// TIA Portal V18 export
// export: Created 2026-06-07T17:38:18.1714676Z, ExportSetting WithDefaults, DisplayName Totally Integrated Automation Portal, DisplayVersion V18, DisplayName TIA Portal Openness, DisplayVersion V18, DisplayName TIA Portal Version Control Interface, DisplayVersion V18, DisplayName STEP 7 Professional, DisplayVersion V18, DisplayName STEP 7 Safety, DisplayVersion V18, DisplayName WinCC Professional, DisplayVersion V18
FUNCTION "FC_HMI_Mirror_PLC1" : Void   // FC41, LAD
{ S7_Optimized_Access := 'TRUE' }
VERSION : 0.1
// stored: AutoNumber true, IsIECCheckEnabled false, SetENOAutomatically false, UDAEnableTagReadback false
BEGIN

REGION Network 1: Mirror AI_V3230_Nuoc_Bon1
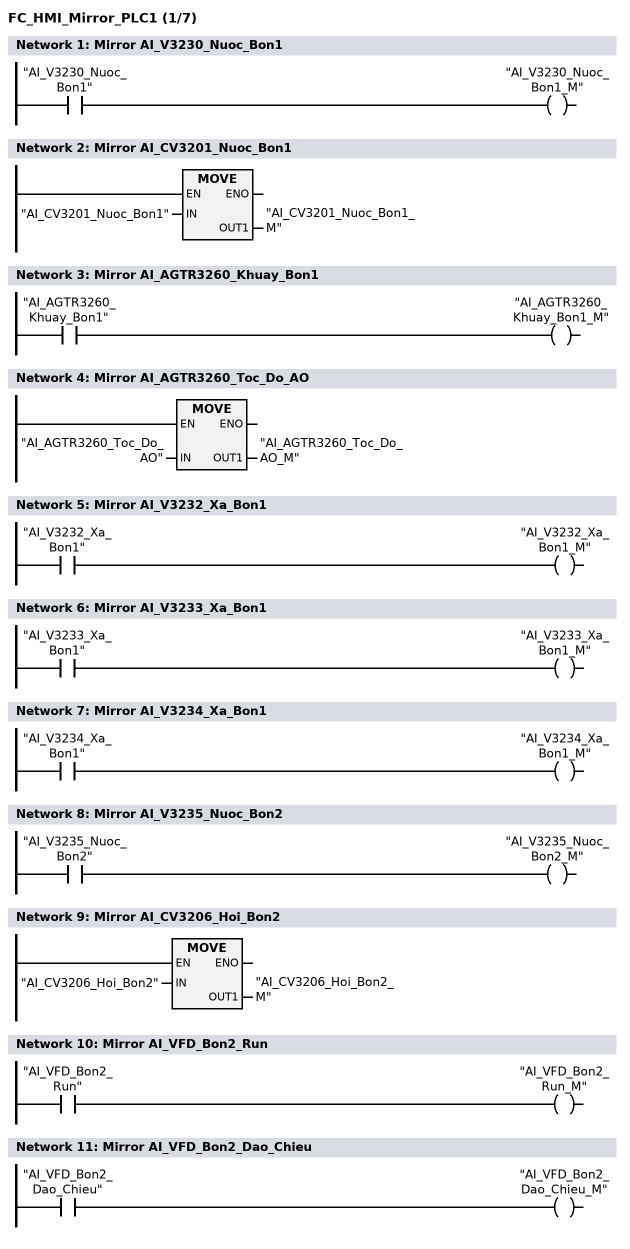
   RUNG wire#powerrail
      Contact( "AI_V3230_Nuoc_Bon1" )
      Coil( "AI_V3230_Nuoc_Bon1_M" )
   END_RUNG
   // the same network as SCL:
   "AI_V3230_Nuoc_Bon1_M" := "AI_V3230_Nuoc_Bon1";
END_REGION

REGION Network 2: Mirror AI_CV3201_Nuoc_Bon1
   RUNG wire#powerrail
      { S7_GenerateENO := "TRUE" } Move(in := "AI_CV3201_Nuoc_Bon1", out1 => "AI_CV3201_Nuoc_Bon1_M")
   END_RUNG
   // the same network as SCL:
   "AI_CV3201_Nuoc_Bon1_M" := "AI_CV3201_Nuoc_Bon1";
END_REGION

REGION Network 3: Mirror AI_AGTR3260_Khuay_Bon1
   RUNG wire#powerrail
      Contact( "AI_AGTR3260_Khuay_Bon1" )
      Coil( "AI_AGTR3260_Khuay_Bon1_M" )
   END_RUNG
   // the same network as SCL:
   "AI_AGTR3260_Khuay_Bon1_M" := "AI_AGTR3260_Khuay_Bon1";
END_REGION

REGION Network 4: Mirror AI_AGTR3260_Toc_Do_AO
   RUNG wire#powerrail
      { S7_GenerateENO := "TRUE" } Move(in := "AI_AGTR3260_Toc_Do_AO", out1 => "AI_AGTR3260_Toc_Do_AO_M")
   END_RUNG
   // the same network as SCL:
   "AI_AGTR3260_Toc_Do_AO_M" := "AI_AGTR3260_Toc_Do_AO";
END_REGION

REGION Network 5: Mirror AI_V3232_Xa_Bon1
   RUNG wire#powerrail
      Contact( "AI_V3232_Xa_Bon1" )
      Coil( "AI_V3232_Xa_Bon1_M" )
   END_RUNG
   // the same network as SCL:
   "AI_V3232_Xa_Bon1_M" := "AI_V3232_Xa_Bon1";
END_REGION

REGION Network 6: Mirror AI_V3233_Xa_Bon1
   RUNG wire#powerrail
      Contact( "AI_V3233_Xa_Bon1" )
      Coil( "AI_V3233_Xa_Bon1_M" )
   END_RUNG
   // the same network as SCL:
   "AI_V3233_Xa_Bon1_M" := "AI_V3233_Xa_Bon1";
END_REGION

REGION Network 7: Mirror AI_V3234_Xa_Bon1
   RUNG wire#powerrail
      Contact( "AI_V3234_Xa_Bon1" )
      Coil( "AI_V3234_Xa_Bon1_M" )
   END_RUNG
   // the same network as SCL:
   "AI_V3234_Xa_Bon1_M" := "AI_V3234_Xa_Bon1";
END_REGION

REGION Network 8: Mirror AI_V3235_Nuoc_Bon2
   RUNG wire#powerrail
      Contact( "AI_V3235_Nuoc_Bon2" )
      Coil( "AI_V3235_Nuoc_Bon2_M" )
   END_RUNG
   // the same network as SCL:
   "AI_V3235_Nuoc_Bon2_M" := "AI_V3235_Nuoc_Bon2";
END_REGION

REGION Network 9: Mirror AI_CV3206_Hoi_Bon2
   RUNG wire#powerrail
      { S7_GenerateENO := "TRUE" } Move(in := "AI_CV3206_Hoi_Bon2", out1 => "AI_CV3206_Hoi_Bon2_M")
   END_RUNG
   // the same network as SCL:
   "AI_CV3206_Hoi_Bon2_M" := "AI_CV3206_Hoi_Bon2";
END_REGION

REGION Network 10: Mirror AI_VFD_Bon2_Run
   RUNG wire#powerrail
      Contact( "AI_VFD_Bon2_Run" )
      Coil( "AI_VFD_Bon2_Run_M" )
   END_RUNG
   // the same network as SCL:
   "AI_VFD_Bon2_Run_M" := "AI_VFD_Bon2_Run";
END_REGION

REGION Network 11: Mirror AI_VFD_Bon2_Dao_Chieu
   RUNG wire#powerrail
      Contact( "AI_VFD_Bon2_Dao_Chieu" )
      Coil( "AI_VFD_Bon2_Dao_Chieu_M" )
   END_RUNG
   // the same network as SCL:
   "AI_VFD_Bon2_Dao_Chieu_M" := "AI_VFD_Bon2_Dao_Chieu";
END_REGION

REGION Network 12: Mirror AI_VFD_Bon2_Toc_Do_AO
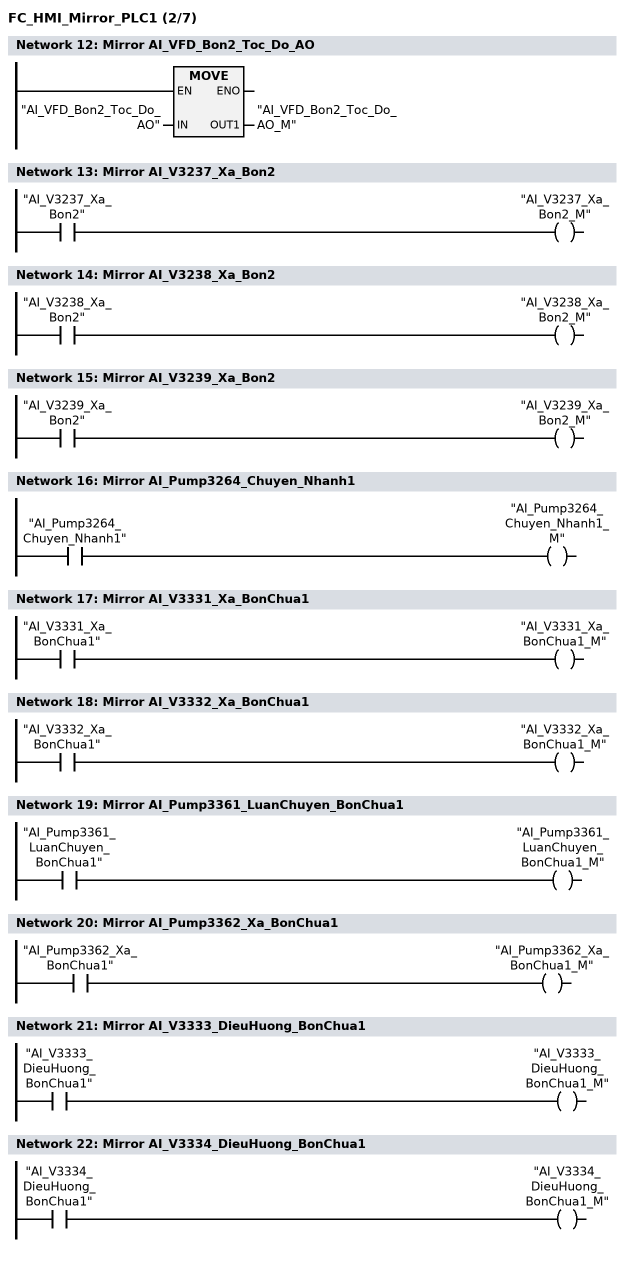
   RUNG wire#powerrail
      { S7_GenerateENO := "TRUE" } Move(in := "AI_VFD_Bon2_Toc_Do_AO", out1 => "AI_VFD_Bon2_Toc_Do_AO_M")
   END_RUNG
   // the same network as SCL:
   "AI_VFD_Bon2_Toc_Do_AO_M" := "AI_VFD_Bon2_Toc_Do_AO";
END_REGION

REGION Network 13: Mirror AI_V3237_Xa_Bon2
   RUNG wire#powerrail
      Contact( "AI_V3237_Xa_Bon2" )
      Coil( "AI_V3237_Xa_Bon2_M" )
   END_RUNG
   // the same network as SCL:
   "AI_V3237_Xa_Bon2_M" := "AI_V3237_Xa_Bon2";
END_REGION

REGION Network 14: Mirror AI_V3238_Xa_Bon2
   RUNG wire#powerrail
      Contact( "AI_V3238_Xa_Bon2" )
      Coil( "AI_V3238_Xa_Bon2_M" )
   END_RUNG
   // the same network as SCL:
   "AI_V3238_Xa_Bon2_M" := "AI_V3238_Xa_Bon2";
END_REGION

REGION Network 15: Mirror AI_V3239_Xa_Bon2
   RUNG wire#powerrail
      Contact( "AI_V3239_Xa_Bon2" )
      Coil( "AI_V3239_Xa_Bon2_M" )
   END_RUNG
   // the same network as SCL:
   "AI_V3239_Xa_Bon2_M" := "AI_V3239_Xa_Bon2";
END_REGION

REGION Network 16: Mirror AI_Pump3264_Chuyen_Nhanh1
   RUNG wire#powerrail
      Contact( "AI_Pump3264_Chuyen_Nhanh1" )
      Coil( "AI_Pump3264_Chuyen_Nhanh1_M" )
   END_RUNG
   // the same network as SCL:
   "AI_Pump3264_Chuyen_Nhanh1_M" := "AI_Pump3264_Chuyen_Nhanh1";
END_REGION

REGION Network 17: Mirror AI_V3331_Xa_BonChua1
   RUNG wire#powerrail
      Contact( "AI_V3331_Xa_BonChua1" )
      Coil( "AI_V3331_Xa_BonChua1_M" )
   END_RUNG
   // the same network as SCL:
   "AI_V3331_Xa_BonChua1_M" := "AI_V3331_Xa_BonChua1";
END_REGION

REGION Network 18: Mirror AI_V3332_Xa_BonChua1
   RUNG wire#powerrail
      Contact( "AI_V3332_Xa_BonChua1" )
      Coil( "AI_V3332_Xa_BonChua1_M" )
   END_RUNG
   // the same network as SCL:
   "AI_V3332_Xa_BonChua1_M" := "AI_V3332_Xa_BonChua1";
END_REGION

REGION Network 19: Mirror AI_Pump3361_LuanChuyen_BonChua1
   RUNG wire#powerrail
      Contact( "AI_Pump3361_LuanChuyen_BonChua1" )
      Coil( "AI_Pump3361_LuanChuyen_BonChua1_M" )
   END_RUNG
   // the same network as SCL:
   "AI_Pump3361_LuanChuyen_BonChua1_M" := "AI_Pump3361_LuanChuyen_BonChua1";
END_REGION

REGION Network 20: Mirror AI_Pump3362_Xa_BonChua1
   RUNG wire#powerrail
      Contact( "AI_Pump3362_Xa_BonChua1" )
      Coil( "AI_Pump3362_Xa_BonChua1_M" )
   END_RUNG
   // the same network as SCL:
   "AI_Pump3362_Xa_BonChua1_M" := "AI_Pump3362_Xa_BonChua1";
END_REGION

REGION Network 21: Mirror AI_V3333_DieuHuong_BonChua1
   RUNG wire#powerrail
      Contact( "AI_V3333_DieuHuong_BonChua1" )
      Coil( "AI_V3333_DieuHuong_BonChua1_M" )
   END_RUNG
   // the same network as SCL:
   "AI_V3333_DieuHuong_BonChua1_M" := "AI_V3333_DieuHuong_BonChua1";
END_REGION

REGION Network 22: Mirror AI_V3334_DieuHuong_BonChua1
   RUNG wire#powerrail
      Contact( "AI_V3334_DieuHuong_BonChua1" )
      Coil( "AI_V3334_DieuHuong_BonChua1_M" )
   END_RUNG
   // the same network as SCL:
   "AI_V3334_DieuHuong_BonChua1_M" := "AI_V3334_DieuHuong_BonChua1";
END_REGION

REGION Network 23: Mirror AI_V3335_DieuHuong_BonChua1
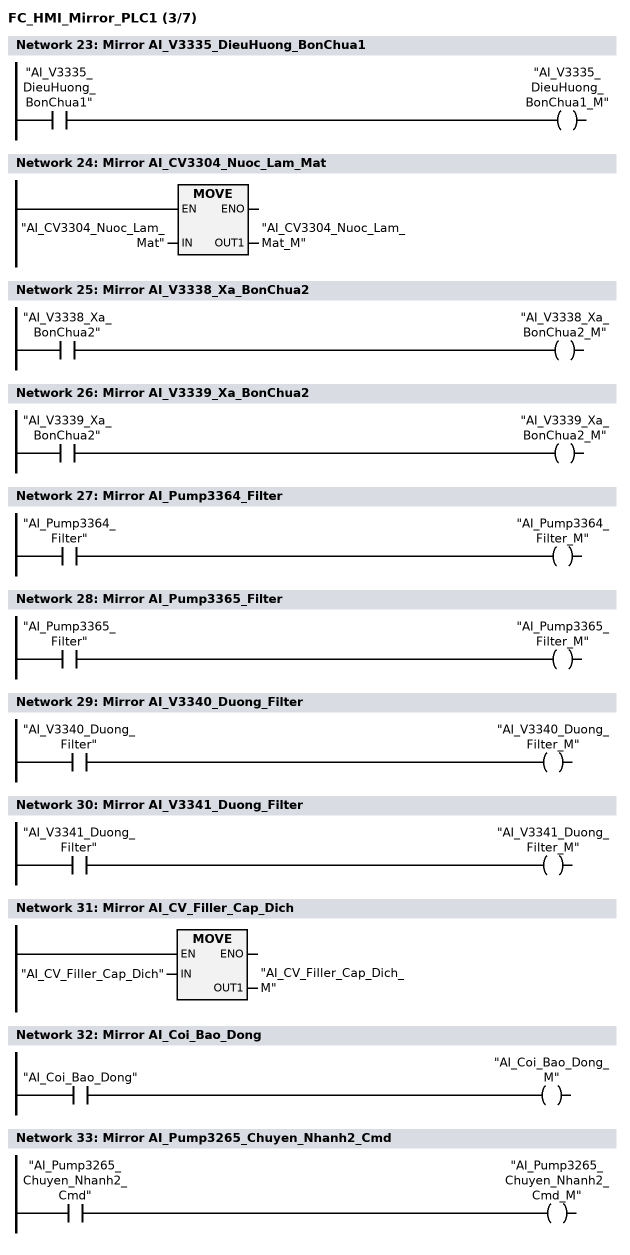
   RUNG wire#powerrail
      Contact( "AI_V3335_DieuHuong_BonChua1" )
      Coil( "AI_V3335_DieuHuong_BonChua1_M" )
   END_RUNG
   // the same network as SCL:
   "AI_V3335_DieuHuong_BonChua1_M" := "AI_V3335_DieuHuong_BonChua1";
END_REGION

REGION Network 24: Mirror AI_CV3304_Nuoc_Lam_Mat
   RUNG wire#powerrail
      { S7_GenerateENO := "TRUE" } Move(in := "AI_CV3304_Nuoc_Lam_Mat", out1 => "AI_CV3304_Nuoc_Lam_Mat_M")
   END_RUNG
   // the same network as SCL:
   "AI_CV3304_Nuoc_Lam_Mat_M" := "AI_CV3304_Nuoc_Lam_Mat";
END_REGION

REGION Network 25: Mirror AI_V3338_Xa_BonChua2
   RUNG wire#powerrail
      Contact( "AI_V3338_Xa_BonChua2" )
      Coil( "AI_V3338_Xa_BonChua2_M" )
   END_RUNG
   // the same network as SCL:
   "AI_V3338_Xa_BonChua2_M" := "AI_V3338_Xa_BonChua2";
END_REGION

REGION Network 26: Mirror AI_V3339_Xa_BonChua2
   RUNG wire#powerrail
      Contact( "AI_V3339_Xa_BonChua2" )
      Coil( "AI_V3339_Xa_BonChua2_M" )
   END_RUNG
   // the same network as SCL:
   "AI_V3339_Xa_BonChua2_M" := "AI_V3339_Xa_BonChua2";
END_REGION

REGION Network 27: Mirror AI_Pump3364_Filter
   RUNG wire#powerrail
      Contact( "AI_Pump3364_Filter" )
      Coil( "AI_Pump3364_Filter_M" )
   END_RUNG
   // the same network as SCL:
   "AI_Pump3364_Filter_M" := "AI_Pump3364_Filter";
END_REGION

REGION Network 28: Mirror AI_Pump3365_Filter
   RUNG wire#powerrail
      Contact( "AI_Pump3365_Filter" )
      Coil( "AI_Pump3365_Filter_M" )
   END_RUNG
   // the same network as SCL:
   "AI_Pump3365_Filter_M" := "AI_Pump3365_Filter";
END_REGION

REGION Network 29: Mirror AI_V3340_Duong_Filter
   RUNG wire#powerrail
      Contact( "AI_V3340_Duong_Filter" )
      Coil( "AI_V3340_Duong_Filter_M" )
   END_RUNG
   // the same network as SCL:
   "AI_V3340_Duong_Filter_M" := "AI_V3340_Duong_Filter";
END_REGION

REGION Network 30: Mirror AI_V3341_Duong_Filter
   RUNG wire#powerrail
      Contact( "AI_V3341_Duong_Filter" )
      Coil( "AI_V3341_Duong_Filter_M" )
   END_RUNG
   // the same network as SCL:
   "AI_V3341_Duong_Filter_M" := "AI_V3341_Duong_Filter";
END_REGION

REGION Network 31: Mirror AI_CV_Filler_Cap_Dich
   RUNG wire#powerrail
      { S7_GenerateENO := "TRUE" } Move(in := "AI_CV_Filler_Cap_Dich", out1 => "AI_CV_Filler_Cap_Dich_M")
   END_RUNG
   // the same network as SCL:
   "AI_CV_Filler_Cap_Dich_M" := "AI_CV_Filler_Cap_Dich";
END_REGION

REGION Network 32: Mirror AI_Coi_Bao_Dong
   RUNG wire#powerrail
      Contact( "AI_Coi_Bao_Dong" )
      Coil( "AI_Coi_Bao_Dong_M" )
   END_RUNG
   // the same network as SCL:
   "AI_Coi_Bao_Dong_M" := "AI_Coi_Bao_Dong";
END_REGION

REGION Network 33: Mirror AI_Pump3265_Chuyen_Nhanh2_Cmd
   RUNG wire#powerrail
      Contact( "AI_Pump3265_Chuyen_Nhanh2_Cmd" )
      Coil( "AI_Pump3265_Chuyen_Nhanh2_Cmd_M" )
   END_RUNG
   // the same network as SCL:
   "AI_Pump3265_Chuyen_Nhanh2_Cmd_M" := "AI_Pump3265_Chuyen_Nhanh2_Cmd";
END_REGION

REGION Network 34: Mirror AI_VFD_Bon2_Actual_Speed_Feedback
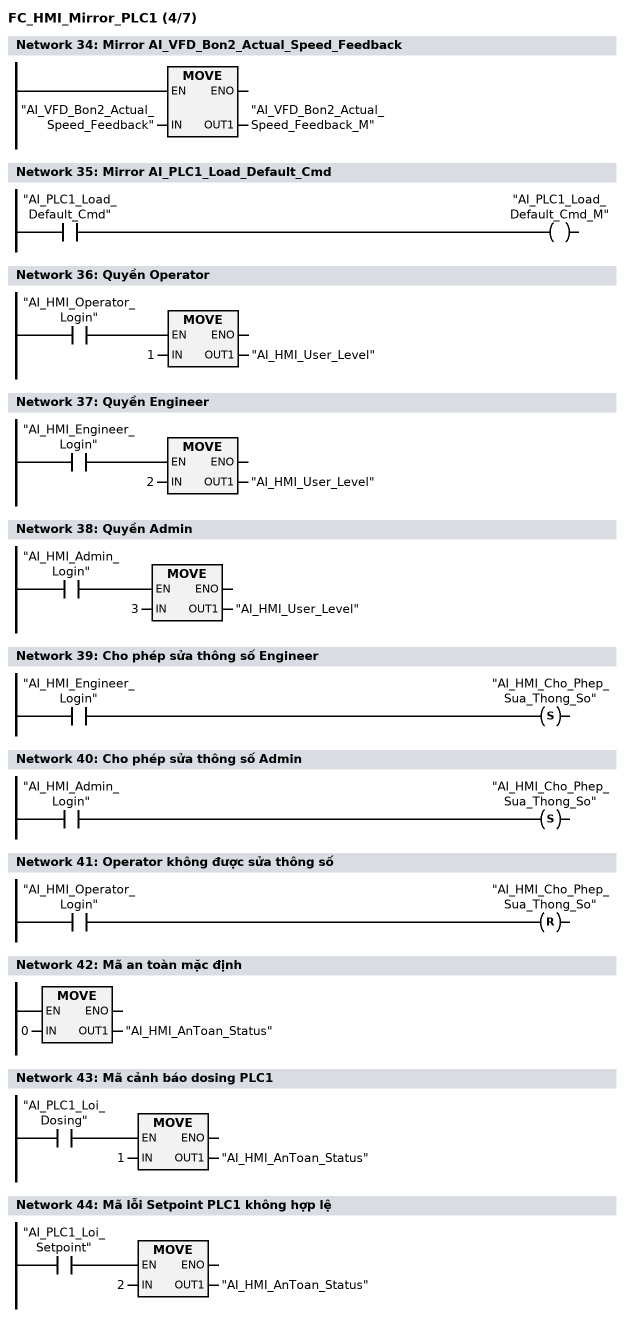
   RUNG wire#powerrail
      { S7_GenerateENO := "TRUE" } Move(in := "AI_VFD_Bon2_Actual_Speed_Feedback", out1 => "AI_VFD_Bon2_Actual_Speed_Feedback_M")
   END_RUNG
   // the same network as SCL:
   "AI_VFD_Bon2_Actual_Speed_Feedback_M" := "AI_VFD_Bon2_Actual_Speed_Feedback";
END_REGION

REGION Network 35: Mirror AI_PLC1_Load_Default_Cmd
   RUNG wire#powerrail
      Contact( "AI_PLC1_Load_Default_Cmd" )
      Coil( "AI_PLC1_Load_Default_Cmd_M" )
   END_RUNG
   // the same network as SCL:
   "AI_PLC1_Load_Default_Cmd_M" := "AI_PLC1_Load_Default_Cmd";
END_REGION

REGION Network 36: Quyền Operator
   RUNG wire#powerrail
      Contact( "AI_HMI_Operator_Login" )
      { S7_GenerateENO := "TRUE" } Move(in := 1, out1 => "AI_HMI_User_Level")
   END_RUNG
   // the same network as SCL:
   IF "AI_HMI_Operator_Login" THEN "AI_HMI_User_Level" := 1; END_IF;
END_REGION

REGION Network 37: Quyền Engineer
   RUNG wire#powerrail
      Contact( "AI_HMI_Engineer_Login" )
      { S7_GenerateENO := "TRUE" } Move(in := 2, out1 => "AI_HMI_User_Level")
   END_RUNG
   // the same network as SCL:
   IF "AI_HMI_Engineer_Login" THEN "AI_HMI_User_Level" := 2; END_IF;
END_REGION

REGION Network 38: Quyền Admin
   RUNG wire#powerrail
      Contact( "AI_HMI_Admin_Login" )
      { S7_GenerateENO := "TRUE" } Move(in := 3, out1 => "AI_HMI_User_Level")
   END_RUNG
   // the same network as SCL:
   IF "AI_HMI_Admin_Login" THEN "AI_HMI_User_Level" := 3; END_IF;
END_REGION

REGION Network 39: Cho phép sửa thông số Engineer
   RUNG wire#powerrail
      Contact( "AI_HMI_Engineer_Login" )
      S_Coil( "AI_HMI_Cho_Phep_Sua_Thong_So" )
   END_RUNG
   // the same network as SCL:
   IF "AI_HMI_Engineer_Login" THEN "AI_HMI_Cho_Phep_Sua_Thong_So" := TRUE; END_IF;
END_REGION

REGION Network 40: Cho phép sửa thông số Admin
   RUNG wire#powerrail
      Contact( "AI_HMI_Admin_Login" )
      S_Coil( "AI_HMI_Cho_Phep_Sua_Thong_So" )
   END_RUNG
   // the same network as SCL:
   IF "AI_HMI_Admin_Login" THEN "AI_HMI_Cho_Phep_Sua_Thong_So" := TRUE; END_IF;
END_REGION

REGION Network 41: Operator không được sửa thông số
   RUNG wire#powerrail
      Contact( "AI_HMI_Operator_Login" )
      R_Coil( "AI_HMI_Cho_Phep_Sua_Thong_So" )
   END_RUNG
   // the same network as SCL:
   IF "AI_HMI_Operator_Login" THEN "AI_HMI_Cho_Phep_Sua_Thong_So" := FALSE; END_IF;
END_REGION

REGION Network 42: Mã an toàn mặc định
   RUNG wire#powerrail
      { S7_GenerateENO := "TRUE" } Move(in := 0, out1 => "AI_HMI_AnToan_Status")
   END_RUNG
   // the same network as SCL:
   "AI_HMI_AnToan_Status" := 0;
END_REGION

REGION Network 43: Mã cảnh báo dosing PLC1
   RUNG wire#powerrail
      Contact( "AI_PLC1_Loi_Dosing" )
      { S7_GenerateENO := "TRUE" } Move(in := 1, out1 => "AI_HMI_AnToan_Status")
   END_RUNG
   // the same network as SCL:
   IF "AI_PLC1_Loi_Dosing" THEN "AI_HMI_AnToan_Status" := 1; END_IF;
END_REGION

REGION Network 44: Mã lỗi Setpoint PLC1 không hợp lệ
   RUNG wire#powerrail
      Contact( "AI_PLC1_Loi_Setpoint" )
      { S7_GenerateENO := "TRUE" } Move(in := 2, out1 => "AI_HMI_AnToan_Status")
   END_RUNG
   // the same network as SCL:
   IF "AI_PLC1_Loi_Setpoint" THEN "AI_HMI_AnToan_Status" := 2; END_IF;
END_REGION

REGION Network 45: Mã lỗi Setpoint Bồn chứa không hợp lệ
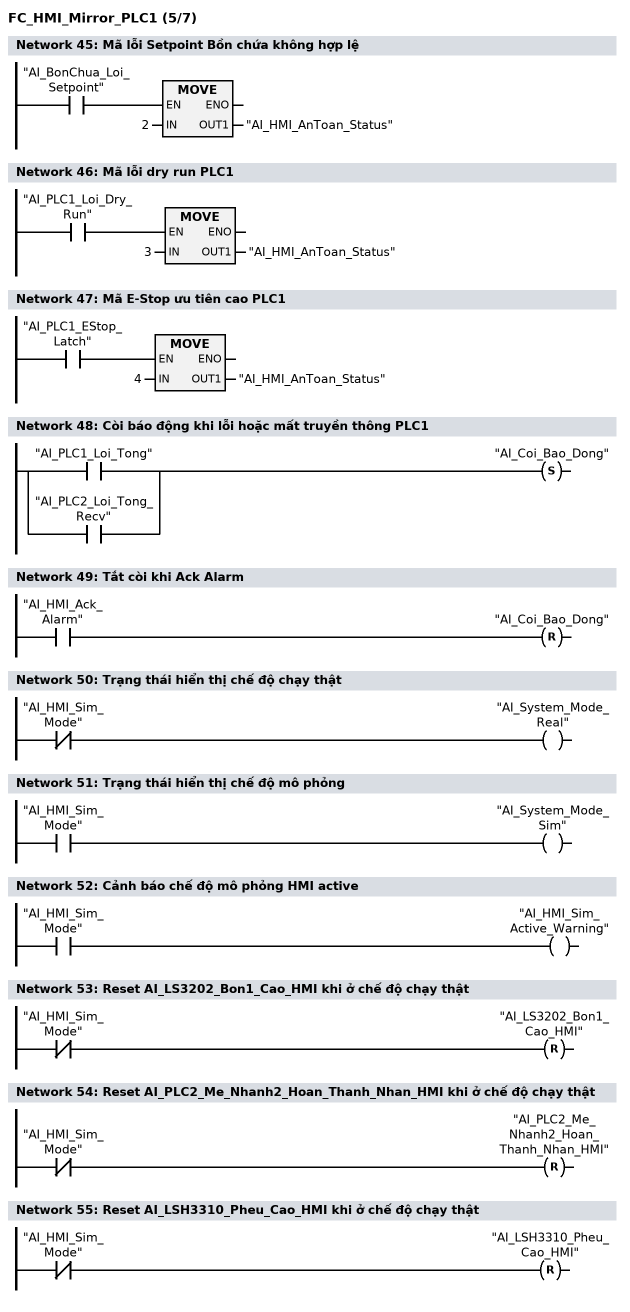
   RUNG wire#powerrail
      Contact( "AI_BonChua_Loi_Setpoint" )
      { S7_GenerateENO := "TRUE" } Move(in := 2, out1 => "AI_HMI_AnToan_Status")
   END_RUNG
   // the same network as SCL:
   IF "AI_BonChua_Loi_Setpoint" THEN "AI_HMI_AnToan_Status" := 2; END_IF;
END_REGION

REGION Network 46: Mã lỗi dry run PLC1
   RUNG wire#powerrail
      Contact( "AI_PLC1_Loi_Dry_Run" )
      { S7_GenerateENO := "TRUE" } Move(in := 3, out1 => "AI_HMI_AnToan_Status")
   END_RUNG
   // the same network as SCL:
   IF "AI_PLC1_Loi_Dry_Run" THEN "AI_HMI_AnToan_Status" := 3; END_IF;
END_REGION

REGION Network 47: Mã E-Stop ưu tiên cao PLC1
   RUNG wire#powerrail
      Contact( "AI_PLC1_EStop_Latch" )
      { S7_GenerateENO := "TRUE" } Move(in := 4, out1 => "AI_HMI_AnToan_Status")
   END_RUNG
   // the same network as SCL:
   IF "AI_PLC1_EStop_Latch" THEN "AI_HMI_AnToan_Status" := 4; END_IF;
END_REGION

REGION Network 48: Còi báo động khi lỗi hoặc mất truyền thông PLC1
   RUNG wire#powerrail
      Contact( "AI_PLC1_Loi_Tong" )
      wire#w1
      S_Coil( "AI_Coi_Bao_Dong" )
   END_RUNG
   RUNG wire#powerrail
      Contact( "AI_PLC2_Loi_Tong_Recv" )
   END_RUNG wire#w1
   // the same network as SCL:
   IF "AI_PLC1_Loi_Tong" OR "AI_PLC2_Loi_Tong_Recv" THEN "AI_Coi_Bao_Dong" := TRUE; END_IF;
END_REGION

REGION Network 49: Tắt còi khi Ack Alarm
   RUNG wire#powerrail
      Contact( "AI_HMI_Ack_Alarm" )
      R_Coil( "AI_Coi_Bao_Dong" )
   END_RUNG
   // the same network as SCL:
   IF "AI_HMI_Ack_Alarm" THEN "AI_Coi_Bao_Dong" := FALSE; END_IF;
END_REGION

REGION Network 50: Trạng thái hiển thị chế độ chạy thật
   RUNG wire#powerrail
      I_Contact( "AI_HMI_Sim_Mode" )
      Coil( "AI_System_Mode_Real" )
   END_RUNG
   // the same network as SCL:
   "AI_System_Mode_Real" := NOT "AI_HMI_Sim_Mode";
END_REGION

REGION Network 51: Trạng thái hiển thị chế độ mô phỏng
   RUNG wire#powerrail
      Contact( "AI_HMI_Sim_Mode" )
      Coil( "AI_System_Mode_Sim" )
   END_RUNG
   // the same network as SCL:
   "AI_System_Mode_Sim" := "AI_HMI_Sim_Mode";
END_REGION

REGION Network 52: Cảnh báo chế độ mô phỏng HMI active
   RUNG wire#powerrail
      Contact( "AI_HMI_Sim_Mode" )
      Coil( "AI_HMI_Sim_Active_Warning" )
   END_RUNG
   // the same network as SCL:
   "AI_HMI_Sim_Active_Warning" := "AI_HMI_Sim_Mode";
END_REGION

REGION Network 53: Reset AI_LS3202_Bon1_Cao_HMI khi ở chế độ chạy thật
   RUNG wire#powerrail
      I_Contact( "AI_HMI_Sim_Mode" )
      R_Coil( "AI_LS3202_Bon1_Cao_HMI" )
   END_RUNG
   // the same network as SCL:
   IF NOT "AI_HMI_Sim_Mode" THEN "AI_LS3202_Bon1_Cao_HMI" := FALSE; END_IF;
END_REGION

REGION Network 54: Reset AI_PLC2_Me_Nhanh2_Hoan_Thanh_Nhan_HMI khi ở chế độ chạy thật
   RUNG wire#powerrail
      I_Contact( "AI_HMI_Sim_Mode" )
      R_Coil( "AI_PLC2_Me_Nhanh2_Hoan_Thanh_Nhan_HMI" )
   END_RUNG
   // the same network as SCL:
   IF NOT "AI_HMI_Sim_Mode" THEN "AI_PLC2_Me_Nhanh2_Hoan_Thanh_Nhan_HMI" := FALSE; END_IF;
END_REGION

REGION Network 55: Reset AI_LSH3310_Pheu_Cao_HMI khi ở chế độ chạy thật
   RUNG wire#powerrail
      I_Contact( "AI_HMI_Sim_Mode" )
      R_Coil( "AI_LSH3310_Pheu_Cao_HMI" )
   END_RUNG
   // the same network as SCL:
   IF NOT "AI_HMI_Sim_Mode" THEN "AI_LSH3310_Pheu_Cao_HMI" := FALSE; END_IF;
END_REGION

REGION Network 56: Reset AI_LSL3311_Pheu_Thap_HMI khi ở chế độ chạy thật
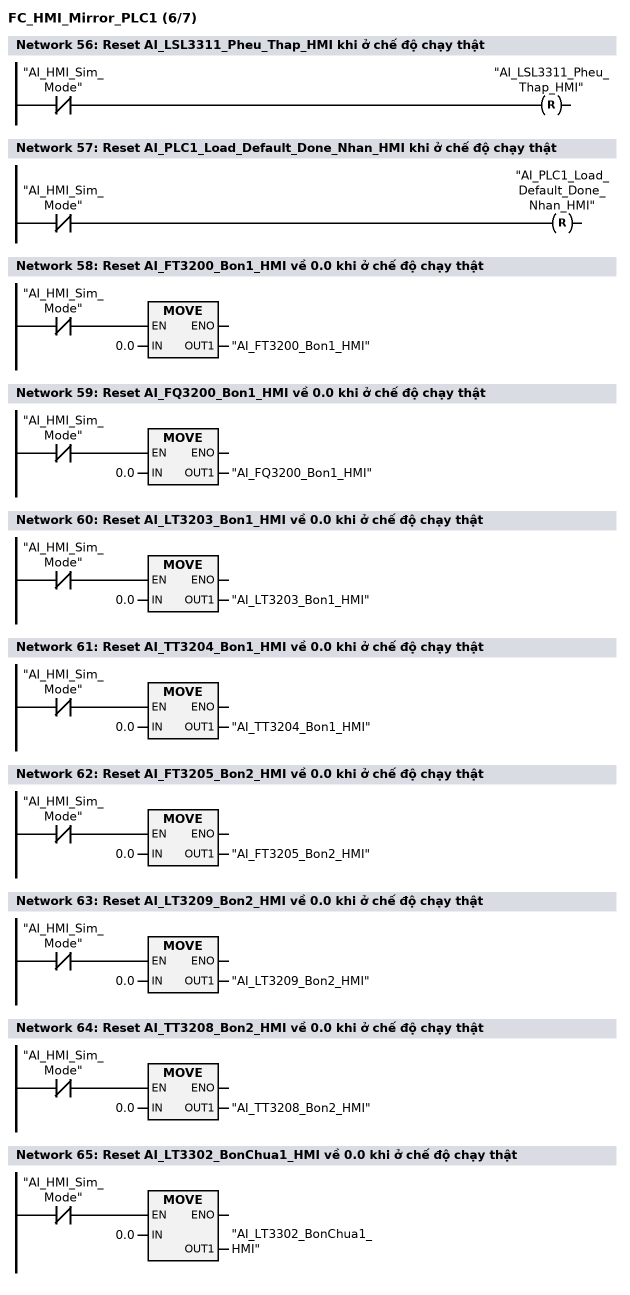
   RUNG wire#powerrail
      I_Contact( "AI_HMI_Sim_Mode" )
      R_Coil( "AI_LSL3311_Pheu_Thap_HMI" )
   END_RUNG
   // the same network as SCL:
   IF NOT "AI_HMI_Sim_Mode" THEN "AI_LSL3311_Pheu_Thap_HMI" := FALSE; END_IF;
END_REGION

REGION Network 57: Reset AI_PLC1_Load_Default_Done_Nhan_HMI khi ở chế độ chạy thật
   RUNG wire#powerrail
      I_Contact( "AI_HMI_Sim_Mode" )
      R_Coil( "AI_PLC1_Load_Default_Done_Nhan_HMI" )
   END_RUNG
   // the same network as SCL:
   IF NOT "AI_HMI_Sim_Mode" THEN "AI_PLC1_Load_Default_Done_Nhan_HMI" := FALSE; END_IF;
END_REGION

REGION Network 58: Reset AI_FT3200_Bon1_HMI về 0.0 khi ở chế độ chạy thật
   RUNG wire#powerrail
      I_Contact( "AI_HMI_Sim_Mode" )
      { S7_GenerateENO := "TRUE" } Move(in := 0.0, out1 => "AI_FT3200_Bon1_HMI")
   END_RUNG
   // the same network as SCL:
   IF NOT "AI_HMI_Sim_Mode" THEN "AI_FT3200_Bon1_HMI" := 0.0; END_IF;
END_REGION

REGION Network 59: Reset AI_FQ3200_Bon1_HMI về 0.0 khi ở chế độ chạy thật
   RUNG wire#powerrail
      I_Contact( "AI_HMI_Sim_Mode" )
      { S7_GenerateENO := "TRUE" } Move(in := 0.0, out1 => "AI_FQ3200_Bon1_HMI")
   END_RUNG
   // the same network as SCL:
   IF NOT "AI_HMI_Sim_Mode" THEN "AI_FQ3200_Bon1_HMI" := 0.0; END_IF;
END_REGION

REGION Network 60: Reset AI_LT3203_Bon1_HMI về 0.0 khi ở chế độ chạy thật
   RUNG wire#powerrail
      I_Contact( "AI_HMI_Sim_Mode" )
      { S7_GenerateENO := "TRUE" } Move(in := 0.0, out1 => "AI_LT3203_Bon1_HMI")
   END_RUNG
   // the same network as SCL:
   IF NOT "AI_HMI_Sim_Mode" THEN "AI_LT3203_Bon1_HMI" := 0.0; END_IF;
END_REGION

REGION Network 61: Reset AI_TT3204_Bon1_HMI về 0.0 khi ở chế độ chạy thật
   RUNG wire#powerrail
      I_Contact( "AI_HMI_Sim_Mode" )
      { S7_GenerateENO := "TRUE" } Move(in := 0.0, out1 => "AI_TT3204_Bon1_HMI")
   END_RUNG
   // the same network as SCL:
   IF NOT "AI_HMI_Sim_Mode" THEN "AI_TT3204_Bon1_HMI" := 0.0; END_IF;
END_REGION

REGION Network 62: Reset AI_FT3205_Bon2_HMI về 0.0 khi ở chế độ chạy thật
   RUNG wire#powerrail
      I_Contact( "AI_HMI_Sim_Mode" )
      { S7_GenerateENO := "TRUE" } Move(in := 0.0, out1 => "AI_FT3205_Bon2_HMI")
   END_RUNG
   // the same network as SCL:
   IF NOT "AI_HMI_Sim_Mode" THEN "AI_FT3205_Bon2_HMI" := 0.0; END_IF;
END_REGION

REGION Network 63: Reset AI_LT3209_Bon2_HMI về 0.0 khi ở chế độ chạy thật
   RUNG wire#powerrail
      I_Contact( "AI_HMI_Sim_Mode" )
      { S7_GenerateENO := "TRUE" } Move(in := 0.0, out1 => "AI_LT3209_Bon2_HMI")
   END_RUNG
   // the same network as SCL:
   IF NOT "AI_HMI_Sim_Mode" THEN "AI_LT3209_Bon2_HMI" := 0.0; END_IF;
END_REGION

REGION Network 64: Reset AI_TT3208_Bon2_HMI về 0.0 khi ở chế độ chạy thật
   RUNG wire#powerrail
      I_Contact( "AI_HMI_Sim_Mode" )
      { S7_GenerateENO := "TRUE" } Move(in := 0.0, out1 => "AI_TT3208_Bon2_HMI")
   END_RUNG
   // the same network as SCL:
   IF NOT "AI_HMI_Sim_Mode" THEN "AI_TT3208_Bon2_HMI" := 0.0; END_IF;
END_REGION

REGION Network 65: Reset AI_LT3302_BonChua1_HMI về 0.0 khi ở chế độ chạy thật
   RUNG wire#powerrail
      I_Contact( "AI_HMI_Sim_Mode" )
      { S7_GenerateENO := "TRUE" } Move(in := 0.0, out1 => "AI_LT3302_BonChua1_HMI")
   END_RUNG
   // the same network as SCL:
   IF NOT "AI_HMI_Sim_Mode" THEN "AI_LT3302_BonChua1_HMI" := 0.0; END_IF;
END_REGION

REGION Network 66: Reset AI_TT3301_BonChua1_HMI về 0.0 khi ở chế độ chạy thật
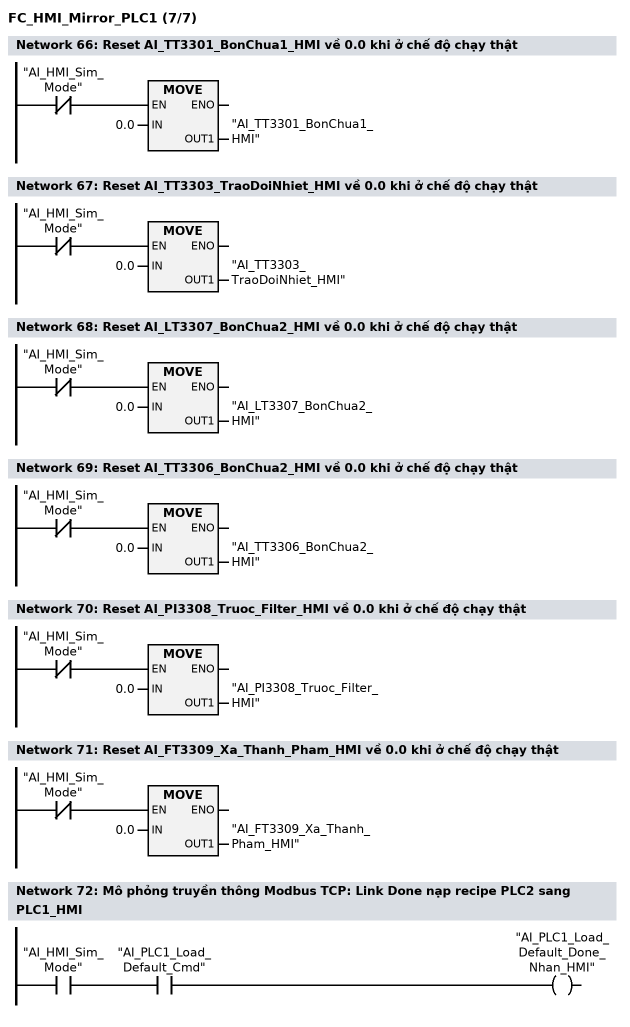
   RUNG wire#powerrail
      I_Contact( "AI_HMI_Sim_Mode" )
      { S7_GenerateENO := "TRUE" } Move(in := 0.0, out1 => "AI_TT3301_BonChua1_HMI")
   END_RUNG
   // the same network as SCL:
   IF NOT "AI_HMI_Sim_Mode" THEN "AI_TT3301_BonChua1_HMI" := 0.0; END_IF;
END_REGION

REGION Network 67: Reset AI_TT3303_TraoDoiNhiet_HMI về 0.0 khi ở chế độ chạy thật
   RUNG wire#powerrail
      I_Contact( "AI_HMI_Sim_Mode" )
      { S7_GenerateENO := "TRUE" } Move(in := 0.0, out1 => "AI_TT3303_TraoDoiNhiet_HMI")
   END_RUNG
   // the same network as SCL:
   IF NOT "AI_HMI_Sim_Mode" THEN "AI_TT3303_TraoDoiNhiet_HMI" := 0.0; END_IF;
END_REGION

REGION Network 68: Reset AI_LT3307_BonChua2_HMI về 0.0 khi ở chế độ chạy thật
   RUNG wire#powerrail
      I_Contact( "AI_HMI_Sim_Mode" )
      { S7_GenerateENO := "TRUE" } Move(in := 0.0, out1 => "AI_LT3307_BonChua2_HMI")
   END_RUNG
   // the same network as SCL:
   IF NOT "AI_HMI_Sim_Mode" THEN "AI_LT3307_BonChua2_HMI" := 0.0; END_IF;
END_REGION

REGION Network 69: Reset AI_TT3306_BonChua2_HMI về 0.0 khi ở chế độ chạy thật
   RUNG wire#powerrail
      I_Contact( "AI_HMI_Sim_Mode" )
      { S7_GenerateENO := "TRUE" } Move(in := 0.0, out1 => "AI_TT3306_BonChua2_HMI")
   END_RUNG
   // the same network as SCL:
   IF NOT "AI_HMI_Sim_Mode" THEN "AI_TT3306_BonChua2_HMI" := 0.0; END_IF;
END_REGION

REGION Network 70: Reset AI_PI3308_Truoc_Filter_HMI về 0.0 khi ở chế độ chạy thật
   RUNG wire#powerrail
      I_Contact( "AI_HMI_Sim_Mode" )
      { S7_GenerateENO := "TRUE" } Move(in := 0.0, out1 => "AI_PI3308_Truoc_Filter_HMI")
   END_RUNG
   // the same network as SCL:
   IF NOT "AI_HMI_Sim_Mode" THEN "AI_PI3308_Truoc_Filter_HMI" := 0.0; END_IF;
END_REGION

REGION Network 71: Reset AI_FT3309_Xa_Thanh_Pham_HMI về 0.0 khi ở chế độ chạy thật
   RUNG wire#powerrail
      I_Contact( "AI_HMI_Sim_Mode" )
      { S7_GenerateENO := "TRUE" } Move(in := 0.0, out1 => "AI_FT3309_Xa_Thanh_Pham_HMI")
   END_RUNG
   // the same network as SCL:
   IF NOT "AI_HMI_Sim_Mode" THEN "AI_FT3309_Xa_Thanh_Pham_HMI" := 0.0; END_IF;
END_REGION

REGION Network 72: Mô phỏng truyền thông Modbus TCP: Link Done nạp recipe PLC2 sang PLC1_HMI
   RUNG wire#powerrail
      Contact( "AI_HMI_Sim_Mode" )
      Contact( "AI_PLC1_Load_Default_Cmd" )
      Coil( "AI_PLC1_Load_Default_Done_Nhan_HMI" )
   END_RUNG
   // the same network as SCL:
   "AI_PLC1_Load_Default_Done_Nhan_HMI" := "AI_HMI_Sim_Mode" AND "AI_PLC1_Load_Default_Cmd";
END_REGION
END_FUNCTION
